RoboDK station: kuka_station.rdk

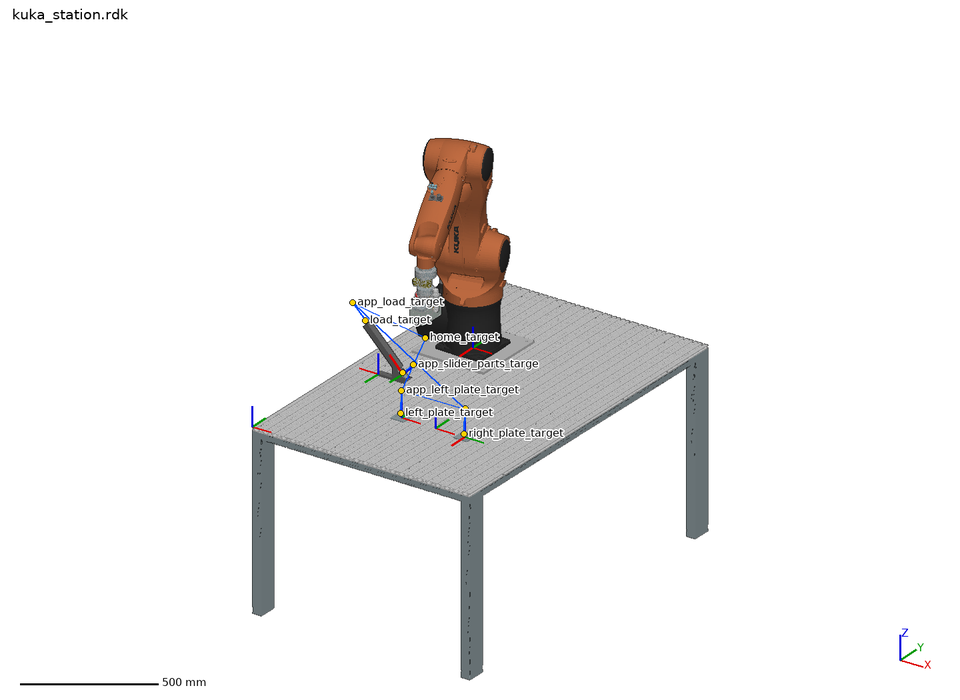
[picture v0: the station drawn from its stored meshes, robots at their saved joint values, targets as dots, program paths as lines]
Station kuka_station (saved by RoboDK 5.9.4). Poses are relative to the parent item; angles as X-Y-Z fixed-axis rotations.
  - frame table_frame at (0, 0, 0) mm
    - object table_object at (0, 0, 0) mm, size 960.1 x 1500 x 750 mm, geometry from table_object.sld
    - target home_target (Cartesian target) at (442.65, 459.31, 297.54) mm, rotated rx 180 ry 0 rz 0 deg; joints [72.96, -71.7, 99.726, 0, 61.974, -64.04] of KUKA KR 6 R900 sixx
    - target left_plate_target (Cartesian target) at (396.2, 370.66, 15.48) mm, rotated rx 180 ry 0 rz 0 deg; joints [79.374, -42.497, 97.48, 0, 35.017, -53.626] of KUKA KR 6 R900 sixx
    - target app_left_plate_target (Cartesian target) at (399.97, 369.91, 110.08) mm, rotated rx 179.99 ry 0 rz 0 deg; joints [79.05, -50.88, 96.36, -180, -44.51, 122.05] of KUKA KR 6 R900 sixx
    - target right_plate_target (Cartesian target) at (679.4, 366.2, 15) mm, rotated rx 180 ry 0 rz 90 deg; joints [57.37, -32.351, 75.287, 0, 47.064, 14.37] of KUKA KR 6 R900 sixx
    - target app_right_plate_target (Cartesian target) at (680, 370.02, 115) mm, rotated rx 180 ry 0.01 rz 93.97 deg; joints [57.169, -40.175, 74.909, -179.995, -55.257, 194.139] of KUKA KR 6 R900 sixx
    - target app_slider_parts_target (Cartesian target) at (277.47, 617.6, 80.28) mm, rotated rx -180 ry 45 rz 0 deg; joints [55.318, -48.751, 125.854, 46.591, 53.169, -119.743] of KUKA KR 6 R900 sixx
    - target slider_parts_target (Cartesian target) at (231.51, 617.6, 34.32) mm, rotated rx -180 ry 45 rz 0 deg; joints [60.38, -42.96, 128.109, 56.425, 47.544, -127.282] of KUKA KR 6 R900 sixx
    - target app_load_target (Cartesian target) at (10, 619, 254.46) mm, rotated rx -180 ry 44.81 rz 0 deg; joints [91.642, -79.146, 135.737, 62.054, 52.892, -89.36] of KUKA KR 6 R900 sixx
    - target load_target (Cartesian target) at (67.51, 617.5, 199.37) mm, rotated rx 180 ry 45 rz 0 deg; joints [82.698, -70.856, 137.084, 62.361, 52.346, -102.667] of KUKA KR 6 R900 sixx
    - target close_gripper_target (joint target) at (399.98, 369.86, -177.92) mm, rotated rx 179.99 ry -0.01 rz -43 deg; joints [20] of gripper
    - target open_gripper_target (joint target) at (400, 370, -278) mm, rotated rx 180 ry 0 rz -43 deg; joints [50] of gripper
  - frame base_plate_frame at (280, 990, 0) mm, rotated rx 0 ry 0 rz -90 deg
    - object base_plate_object at (0, 0, 0) mm, size 320 x 320 x 10 mm, geometry from base_plate_object.sld
  - frame slider_frame at (125, 617, 0) mm, rotated rx 0 ry 0 rz 180 deg
    - object slider_object at (0, 0, 0) mm, size 198.7 x 26 x 198.7 mm, 1 curves, geometry from slider_object.sld
  - frame slider_parts_frame at (232.7, 617, 30.7) mm, rotated rx 0 ry -45 rz 180 deg
    - object part_object at (-0.42, 0, -0.99) mm, size 40 x 20 x 20 mm, 1 curves, geometry from part_object.sld
  - frame pick_and_drop_frame at (550, 370, 0) mm
  - frame right_frame at (680, 370, 0) mm, rotated rx 0 ry 0 rz -90 deg
    - object right_plate_object at (0, 0, 0) mm, size 60 x 60 x 9 mm, 1 curves, geometry from right_plate_object.sld
  - frame left_frame at (400, 370, 0) mm
    - object left_plate_object at (0, 0, 0) mm, size 60 x 60 x 9 mm, 1 curves, geometry from left_plate_object.sld
  - frame kuka_frame at (280, 990, 0) mm
    - robot KUKA KR 6 R900 sixx: 6 axes, payload 6 kg, reach 901 mm, repeatability 0.03 mm, weight 52 kg
        modified DH rows (alpha deg, a mm, theta deg, d mm): 0, 0, 0, 400; -90, 25, 0, 0; 0, 455, -90, 0; -90, 35, 0, 420; 90, 0, 0, 0; -90, 0, 180, 80
        joint limits [-170, -190, -120, -185, -120, -350] to [170, 45, 156, 185, 120, 350]; home [0, -90, 90, 0, 0, 0]; saved at [72.96, -71.7, 99.726, 0, 61.974, -60.04]
      - robot gripper: 1 axes
          joint limits [0] to [50]; home [0]; saved at [50]
      - tool gripper_TCP, TCP at (0, 0, 288) mm, rotated rx 0 ry 0 rz 47 deg
  - folder programs
    - program factory_reset (3 instructions, listed below)
    - program close_target (3 instructions, listed below)
    - program open_target (3 instructions, listed below)
  - program main (32 instructions, listed below)
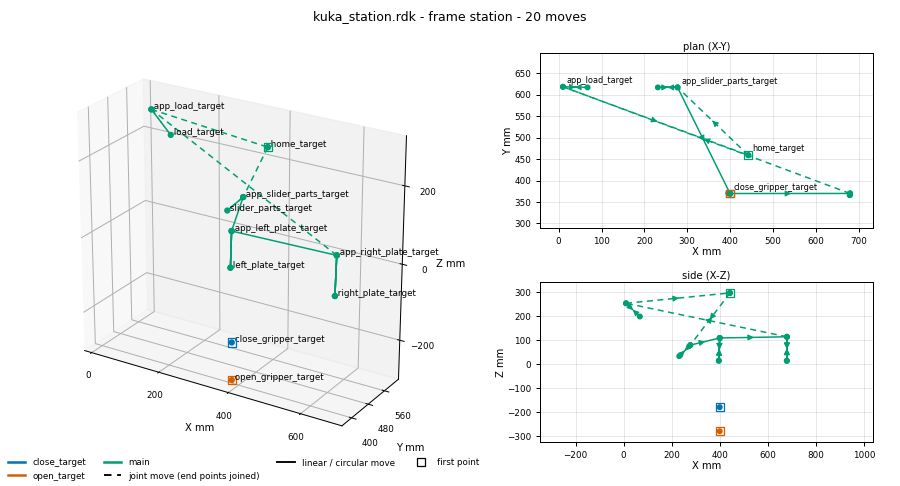
[picture p0: tool path of kuka_station.rdk in frame station, 20 of 20 moves have a stored position in this frame; points joined in program order, loops and branches not executed]

--- program factory_reset (robot KUKA KR 6 R900 sixx) ---
  Replace objects
  Attach to gripper_TCP
  Attach to gripper_TCP

--- program close_target (robot gripper) ---
  Set Ref.: table_frame
  Set Tool: gripper_TCP
  MoveJ (close_t) -> target close_gripper_target

--- program open_target (robot gripper) ---
  Set Ref.: table_frame
  Set Tool: gripper_TCP
  MoveJ (open_t) -> target open_gripper_target

--- program main (robot KUKA KR 6 R900 sixx) ---
  MoveJ (home_target)
  Call factory_reset
  MoveJ (app_slider_parts_target)
  MoveJ (slider_parts_target)
  Call close_target
  Attach to gripper_TCP
  MoveL (app_slider_parts_target)
  MoveL (app_left_plate_target)
  MoveL (left_plate_target)
  Call open_target
  Detach from gripper_TCP
  MoveL (app_left_plate_target)
  MoveL (left_plate_target)
  Call close_target
  Attach to gripper_TCP
  MoveL (app_left_plate_target)
  MoveL (app_right_plate_target)
  MoveL (right_plate_target)
  Call open_target
  Detach from gripper_TCP
  MoveL (app_right_plate_target)
  MoveL (right_plate_target)
  Call close_target
  Attach to gripper_TCP
  MoveL (app_right_plate_target)
  MoveJ (app_load_target)
  MoveJ (load_target)
  Call open_target
  Detach from gripper_TCP
  Call factory_reset
  MoveJ (app_load_target)
  MoveJ (home_target)
